# EPICS autosave request: iocBoot/obsolete/ioc13USBCTR/auto_settings.req
file "USBCTR_settings.req", P=13USBCTR1:
